// TIA Portal V20 export
TYPE "LKinCtrl_typePnPInitTOData"
   STRUCT
      factorBlendingLength : LReal;   // Factor blending length
      orientationDefaults : "LKinCtrl_typePathDynamics";   // Orientation default dynamics
   END_STRUCT;
END_TYPE
